(* IEC 61131-3 sources: stc/stdlib/vendor/schneider, 3 files *)

(* ---- communication.st ---- *)
(* Schneider Electric EcoStruxure -- Communication function blocks *)
(* Modbus and general communication stubs *)

FUNCTION_BLOCK READ_VAR
VAR_INPUT
    ADR         : STRING(32);
    OBJ         : STRING(8);
    NUM         : INT;
    Req         : BOOL;
END_VAR
VAR_OUTPUT
    Done        : BOOL;
    Busy        : BOOL;
    Error       : BOOL;
    Status      : UDINT;
    DataOut     : INT;
END_VAR
END_FUNCTION_BLOCK

FUNCTION_BLOCK WRITE_VAR
VAR_INPUT
    ADR         : STRING(32);
    OBJ         : STRING(8);
    NUM         : INT;
    DataIn      : INT;
    Req         : BOOL;
END_VAR
VAR_OUTPUT
    Done        : BOOL;
    Busy        : BOOL;
    Error       : BOOL;
    Status      : UDINT;
END_VAR
END_FUNCTION_BLOCK

FUNCTION_BLOCK SEND_REQ
VAR_INPUT
    ADR         : STRING(32);
    DataIn      : STRING(255);
    LenIn       : INT;
    Req         : BOOL;
END_VAR
VAR_OUTPUT
    Done        : BOOL;
    Busy        : BOOL;
    Error       : BOOL;
    Status      : UDINT;
    DataOut     : STRING(255);
    LenOut      : INT;
END_VAR
END_FUNCTION_BLOCK

FUNCTION_BLOCK RCV_REQ
VAR_INPUT
    Enable      : BOOL;
    ADR         : STRING(32);
END_VAR
VAR_OUTPUT
    Done        : BOOL;
    Busy        : BOOL;
    Error       : BOOL;
    Status      : UDINT;
    DataOut     : STRING(255);
    LenOut      : INT;
END_VAR
END_FUNCTION_BLOCK

(* ---- motion.st ---- *)
(* Schneider Electric EcoStruxure -- PLCopen Motion Control stubs *)
(* Schneider-specific parameters differ from Beckhoff. *)

(* Schneider AXIS_REF -- different internal structure from Beckhoff *)
TYPE SE_AXIS_REF :
STRUCT
    AxisId      : UDINT;
    AxisState   : INT;
END_STRUCT
END_TYPE

FUNCTION_BLOCK MC_Power
VAR_INPUT
    Axis            : SE_AXIS_REF;
    Enable          : BOOL;
    EnablePositive  : BOOL;
    EnableNegative  : BOOL;
    ControllerMode  : INT;
END_VAR
VAR_OUTPUT
    Status      : BOOL;
    Busy        : BOOL;
    Active      : BOOL;
    Error       : BOOL;
    ErrorID     : UDINT;
END_VAR
END_FUNCTION_BLOCK

FUNCTION_BLOCK MC_MoveAbsolute
VAR_INPUT
    Axis            : SE_AXIS_REF;
    Execute         : BOOL;
    Position        : LREAL;
    Velocity        : LREAL;
    Acceleration    : LREAL;
    Deceleration    : LREAL;
    Jerk            : LREAL;
END_VAR
VAR_OUTPUT
    Done            : BOOL;
    Busy            : BOOL;
    Active          : BOOL;
    CommandAborted  : BOOL;
    Error           : BOOL;
    ErrorID         : UDINT;
END_VAR
END_FUNCTION_BLOCK

FUNCTION_BLOCK MC_Stop
VAR_INPUT
    Axis            : SE_AXIS_REF;
    Execute         : BOOL;
    Deceleration    : LREAL;
    Jerk            : LREAL;
END_VAR
VAR_OUTPUT
    Done            : BOOL;
    Busy            : BOOL;
    Active          : BOOL;
    CommandAborted  : BOOL;
    Error           : BOOL;
    ErrorID         : UDINT;
END_VAR
END_FUNCTION_BLOCK

(* ---- system.st ---- *)
(* Schneider Electric EcoStruxure -- System utility function blocks *)

FUNCTION GetBit : BOOL
VAR_INPUT
    Value       : DWORD;
    BitNum      : INT;
END_VAR
END_FUNCTION

FUNCTION SetBit : DWORD
VAR_INPUT
    Value       : DWORD;
    BitNum      : INT;
    BitValue    : BOOL;
END_VAR
END_FUNCTION

FUNCTION_BLOCK RTC
VAR_INPUT
    EN          : BOOL;
    PDT         : STRING(20);
END_VAR
VAR_OUTPUT
    Q           : BOOL;
    CDT         : STRING(20);
END_VAR
END_FUNCTION_BLOCK
